PROGRAM P_Decorator
VAR
	ErrorString				: STRING;
	stringBuilder			: StringBuilder;
	ErrorNumber				: INT := 1;
	ErrorMessage			: STRING := 'This is my error message';
END_VAR

ErrorString := stringBuilder
					.Clear()
					.Append('Error number: ')
					.Append(INT_TO_STRING(ErrorNumber))
					.Append('. Message: ')
					.Append(ErrorMessage)
					.Append('.')
					.ToString();

END_PROGRAM

(* stored: Version 1.1.0.1, ProductVersion 3.1.4024.12
   POU P_Decorator: Id {8081ffa8-7281-40f4-a0a4-0ae6a00ba4ae}, SpecialFunc None *)
